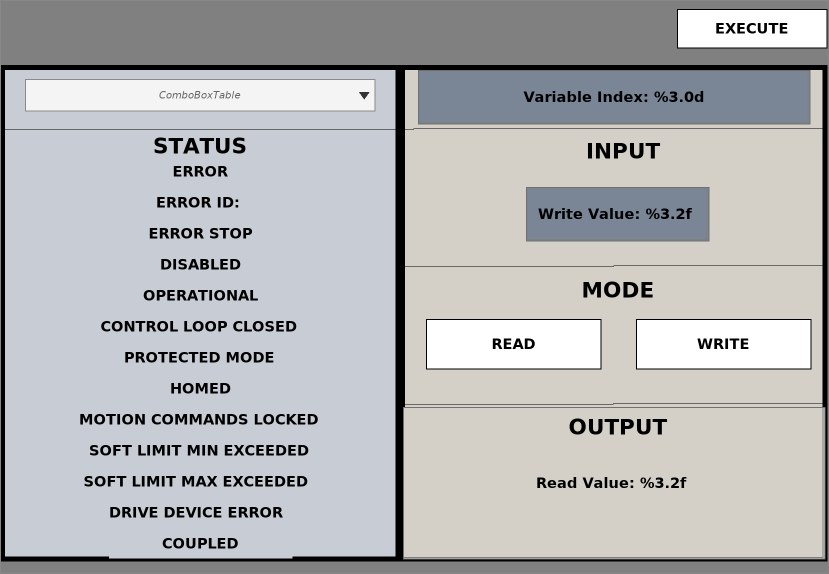
VISUALIZATION parametersScreen  // 829x574
    Rectangle (400,65 427x496)
    Button (403,407 422x152), "Read Value: %3.2f", text variable: multiControl.fValueOut
    RoundedRectangle (677,9 150x39), "EXECUTE", colour toggle: multiControl.bExecute
        toggle multiControl.bExecute
    Rectangle (0,65 400x496)
    Rectangle (109,281 183x29), "OPERATIONAL", colour toggle: multiControl.aStatusVar[4]
    Rectangle (109,374 183x29), "HOMED", colour toggle: multiControl.aStatusVar[7]
    Rectangle (74,312 250x29), "CONTROL LOOP CLOSED", colour toggle: multiControl.aStatusVar[5]
    Button (526,187 183x54), "Write Value: %3.2f", text variable: multiControl.fValueIn
        OnMouseClick: write the text variable via VisuDialogs.Numpad
    Line (0,129) (827,128)
    Line (402,266) (825,265)
    Line (401,404) (825,403)
    RoundedRectangle (426,319 175x50), "READ", colour toggle: multiControl.bReadParam
        toggle multiControl.bReadParam
    RoundedRectangle (636,319 175x50), "WRITE", colour toggle: multiControl.bWriteParam
        toggle multiControl.bWriteParam
    ComboBoxTable (25,79 350x32), variable: multiControl.nMotorControlIndex, data array: multiControl.aMotorSelection
        p3854506369: multiControl.aMotorSelection[INDEX]
    Label (543,275 150x30), "MODE"
    Label (548,136 150x30), "INPUT"
    Label (543,412 150x30), "OUTPUT"
    Label (125,131 150x30), "STATUS"
    Rectangle (109,250 183x29), "DISABLED", colour toggle: multiControl.aStatusVar[3]
    Rectangle (109,219 183x29), "ERROR STOP", colour toggle: multiControl.aStatusVar[2]
    Rectangle (109,188 183x29), "ERROR ID:", colour toggle: multiControl.aMotorActive[1]
    Rectangle (109,157 183x29), "ERROR", colour toggle: multiControl.aStatusVar[1]
    Rectangle (108,343 183x29), "PROTECTED MODE", colour toggle: multiControl.aStatusVar[6]
    Rectangle (64,405 270x29), "MOTION COMMANDS LOCKED", colour toggle: multiControl.aStatusVar[8]
    Rectangle (74,436 250x29), "SOFT LIMIT MIN EXCEEDED", colour toggle: multiControl.aStatusVar[9]
    Rectangle (71,467 250x29), "SOFT LIMIT MAX EXCEEDED", colour toggle: multiControl.aStatusVar[10]
    Rectangle (71,498 250x29), "DRIVE DEVICE ERROR", colour toggle: multiControl.aStatusVar[11]
    Rectangle (109,529 183x29), "COUPLED", colour toggle: multiControl.aStatusVar[12]
    Button (418,70 392x54), "Variable Index: %3.0d", text variable: multiControl.nParameterIndex
        OnMouseClick: write the text variable via VisuDialogs.Numpad
END_VISUALIZATION

(* stored: Version 1.1.0.1, ProductVersion 3.1.4024.13
   Visu parametersScreen: Id {c78001dc-d5fc-4b52-adba-cff16d3db73a} *)
